// TIA Portal V17 export
// export: Created 2025-04-11T04:54:25.0488755Z, ExportSetting WithDefaults, DisplayName Totally Integrated Automation Portal, DisplayVersion V17, DisplayName TIA Portal Openness, DisplayVersion V17, DisplayName TIA Portal Version Control Interface, DisplayVersion V17, DisplayName SINAMICS Startdrive Advanced, DisplayVersion V17, DisplayName SINAMICS Startdrive G130, G150, S120, S150, SINAMICS MV, S210, DisplayVersion V17, DisplayName SINAMICS Startdrive G110M, G120, G120C, G120D, G120P, G115D, DisplayVersion V17, DisplayName STEP 7 Professional, DisplayVersion V17, DisplayName STEP 7 Safety, DisplayVersion V17, DisplayName WinCC Advanced, DisplayVersion V17
TYPE "UDT_Ana_Keep"
// stored: IsFailsafeCompliant false
   STRUCT
      IN_RawHigh : Int;   // 原始值量程上限
      IN_RawLow : Int;   // 原始值量程下限
      IN_EngHigh : Real;   // 工程值量程上限
      IN_EngLow : Real;   // 工程值量程下限
      IN_LLLimit : Real;   // 低低报警限值
      IN_LLimit : Real;   // 低报警限值
      IN_HLimit : Real;   // 高报警限值
      IN_HHLimit : Real;   // 高高报警限值
      IN_DeadBand : Real;   // 报警死区
      IN_AlarmMask : Int;   // 报警屏蔽（0位:高高报警, 1位:高报警, 2位:低报警, 3位:低低报警）
      IN_SensorFaultHigh : Real;   // 传感器故障上限
      IN_SensorFaultLow : Real;   // 传感器故障下限
      IN_ALMEnable : Bool := TRUE;   // 报警使能
      IN_AlarmDelay : Time := T#1S;   // 报警延时
   END_STRUCT;
END_TYPE
